TYPE ST_AutoControlSwitch :
STRUCT
	bExecute: BOOL;
	bDone: BOOL;
	bError: BOOL;
END_STRUCT
END_TYPE

(* stored: Version 1.1.0.1, ProductVersion 3.1.4024.12
   DUT ST_AutoControlSwitch: Id {dab5a2aa-b659-43b5-b399-d0d5c3a7edcf} *)
